# EPICS autosave request: soft_iocs/toaster/iocBoot/ioctoaster/auto_settings.req
file "ao.req", P=$(P)Toast:, D=H:, R=High
file "ao.req", P=$(P)Toast:, D=H:, R=Low
file "sseqRecord_settings.req", P=$(P)Toast:, S=H:Move

file "ao.req", P=$(P)Toast:, D=V:, R=High
file "ao.req", P=$(P)Toast:, D=V:, R=Low
file "sseqRecord_settings.req", P=$(P)Toast:, S=V:Move
